PROGRAM PRG_CASE_InitialiseDataManual
VAR
	fbCase_InitialiseData		: FB_CASE_InitialiseData;
	
	(* Iterator for Init function/method *)
	nOuterIndex				: INT;
	nPackIndex				: INT;
	rTrigDataInit			: R_TRIG;
	bDataInit				: BOOL;
	
	(* Inputs *)	
	bExecute 				: BOOL;	(* set TRUE to move Outers *)
	stCTDateTime			: ST_SYSTEM_DateTime;
	stDoorGuardReject		: ST_RejectItems;
	
	
	(* In/Out *)
	stProductInstruction	: ST_PCM_Status := (sFieldName := 'dupa', nOutersPerCase := 50);
	stCACData 				: ST_CAC_Data;	(* Case Queue *)
	
	(* Outputs *)
	bDone					: BOOL;
	bBusy					: BOOL;
	bDoorReject				: BOOL;
	sRejectCode				: T_MaxString;		
	nMasterListCounter		: INT;	
	bCheckDuplicates		: BOOL;
	
END_VAR

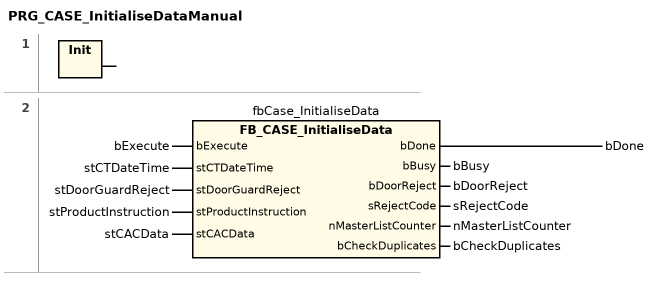
// NETWORK 1
Init();

// NETWORK 2
fbCase_InitialiseData(
    bExecute := bExecute,
    stCTDateTime := stCTDateTime,
    stDoorGuardReject := stDoorGuardReject,
    stProductInstruction := stProductInstruction,
    stCACData := stCACData,
    bBusy => bBusy,
    bDoorReject => bDoorReject,
    sRejectCode => sRejectCode,
    nMasterListCounter => nMasterListCounter,
    bCheckDuplicates => bCheckDuplicates); // FB_CASE_InitialiseData
bDone := fbCase_InitialiseData.bDone;

ACTION Init:

rTrigDataInit(CLK := bDataInit);

IF rTrigDataInit.Q THEN
	
	MEMSET(ADR(stCACData), 16#00, SIZEOF(stCACData));	
	
	stProductInstruction.nOutersPerCase 	:= 50;
	stProductInstruction.nPacksPerOuter		:= 10;
	stProductInstruction.nOpMode			:= 11;
	stProductInstruction.sRetailSKU			:= '1234567';
	stProductInstruction.nAcceptanceLevel 	:= 10;


	stCACData.NumberOfOuters			:= stProductInstruction.nOutersPerCase;
	stCACData.CodingAndTrackingMode		:= stProductInstruction.nOpMode;
	stCACData.RetailSKU					:= stProductInstruction.sRetailSKU;

	FOR nOuterIndex := 1 TO stProductInstruction.nOutersPerCase BY 1 DO
	
	stCACData.Outer[nOuterIndex].Barcode 					:= CONCAT('OUTER_', INT_TO_STRING(nOuterIndex));
	stCACData.Outer[nOuterIndex].NumberOfPacks 				:= stProductInstruction.nPacksPerOuter;
	stCACData.Outer[nOuterIndex].NumberOfLinkedPacks 		:= stProductInstruction.nPacksPerOuter;
	stCACData.Outer[nOuterIndex].AcceptanceLevel 			:= stProductInstruction.nAcceptanceLevel;
	stCACData.Outer[nOuterIndex].CodingAndTrackingMode		:= stProductInstruction.nOpMode;
	stCACData.Outer[nOuterIndex].OuterRejectCode			:= 'OK';
	
		FOR  nPackIndex :=1 TO stProductInstruction.nPacksPerOuter BY 1 DO
			stCACData.Outer[nOuterIndex].PackCode[nPackIndex] 		:= F_CONCAT3(stCACData.Outer[nOuterIndex].Barcode,'_PACK_', INT_TO_STRING(nPackIndex));
			IF nPackIndex = 1 THEN
				stCACData.Outer[nOuterIndex].AggregationCodes[1]	:= stCACData.Outer[nOuterIndex].PackCode[nPackIndex];
			END_IF
			IF nPackIndex = 2 THEN
				stCACData.Outer[nOuterIndex].AggregationCodes[2]	:= stCACData.Outer[nOuterIndex].PackCode[nPackIndex];
			END_IF
			stCACData.Outer[nOuterIndex].PackCodeStatus[nPackIndex].5 	:= TRUE;
			stCACData.Outer[nOuterIndex].PackRejectCode[nPackIndex]		:= 'OK';
		END_FOR
	END_FOR	
	
	stCACData.Outer[3].OuterCodeStatus.5 	:= TRUE;
	stCACData.Outer[4].OuterCodeStatus.5	:= TRUE;
	
END_IF
END_ACTION

END_PROGRAM

(* stored: Version 1.1.0.1
   POU PRG_CASE_InitialiseDataManual: Id {9d983551-81c2-4987-8957-1c8f757bfb69}, SpecialFunc None
   Action Init: Id {cfa3d2a8-acd0-4495-8661-28cac742514f} *)
